// TwinCAT 3 PLC project PRG_PLCHMIManager
// Title: B_PLCHMIManager
// Company: RafalOS
// Author: Rafał Osajda
// ProjectVersion: 0.0.0.23
// ProgramVersion: 3.1.4024.0
// CompilerDefines: VISU_USEWSTRING
// libraries:
//   B_Base, * (RafalOS)
//   B_Base_HMI_Connector, * (RafalOS)
//   B_HMIElements, * (RafalOS)
//   B_HMIManager, * (RafałOS)
//   B_MachineControl_HMI_Connector, * (RafalOS)
//   B_StatesAndModes, * (RafalOS)
//   CmpBitmapPool, * (System)
//   Tc2_Standard, * (Beckhoff Automation GmbH)
//   Tc2_System, * (Beckhoff Automation GmbH)
//   Tc3_Module, * (Beckhoff Automation GmbH)
//   VisuDialogs, * (System)
//   VisuSymbols,3.5.10.0,System
// project tree:
//   / GlobalTextList.TcGTLO, PlcTask.TcTTO, Visualization Manager.TcVMO (not stored), VISU_TASK.TcTTO
//   POUs/ MAIN.TcPOU
//   VISUs/Dialogs/ D_AddRecipe.TcVIS, D_DeleteRecipeCleim.TcVIS
//   VISUs/Frame/ F_Descriptor.TcVIS, F_DiagramState.TcVIS
//   VISUs/Graphics/ ImagePool.TcIPO (not stored)
//   VISUs/Keyboards/ KlawiaturaCyfry.TcVIS, KlawiaturaLitery.TcVIS
//   VISUs/ MainFrame.TcVIS, TextListGlobal.TcTLO, Visualization.TcVIS
//   VISUs/MainMenuFrame/ F_00_MainScreen.TcVIS, F_01_Parameters.TcVIS, F_02_Recipe.TcVIS, F_03_Events.TcVIS, F_04_ChangeMode.TcVIS, F_05_Statistics.TcVIS, F_06_Diagram.TcVIS, F_07_Settings.TcVIS
//   VISUs/MainMenu/ F_MainMenu_00.TcVIS, F_MainMenu_01.TcVIS, F_MainMenu_02.TcVIS, F_MainMenu_03.TcVIS, F_MainMenu_04.TcVIS, F_MainMenu_05.TcVIS, F_MainMenu_06.TcVIS, F_MainMenu_07.TcVIS
//   VISUs/TextListFrame/ TextList_00.TcTLO, TextList_01.TcTLO, TextList_02.TcTLO, TextList_03.TcTLO, TextList_04.TcTLO, TextList_05.TcTLO, TextList_06.TcTLO, TextList_07.TcTLO
// real-time tasks:
//   TASK PlcTask: cycle T#10ms, priority 20, ADS port 350
//   TASK VISU_TASK: cycle T#200000us, priority 30, ADS port 351

CONFIGURATION PRG_PLCHMIManager
    RESOURCE PLC ON TwinCAT3
        TASK PlcTask(INTERVAL := T#10ms, PRIORITY := 20);
        TASK VISU_TASK(INTERVAL := T#200000us, PRIORITY := 30);
        PROGRAM MAIN WITH PlcTask : MAIN;
        PROGRAM VisuElems_Visu_Prg WITH VISU_TASK : VisuElems.Visu_Prg;
    END_RESOURCE
END_CONFIGURATION

// ---- POUs/MAIN.TcPOU
PROGRAM MAIN
VAR
	stDataHMI : ST_HMIManager;
END_VAR

END_PROGRAM

// ---- GlobalTextList.TcGTLO
TEXTLIST GlobalTextList
  338 = '!'
  340 = '"'
  991 = '#'
  344 = '$'
  346 = '%'
  858 = '%d'
  949 = '%s'
  399 = '%s sfdasgfds gkds gow gk wjd k gj dlkg jdl glkd sj g ld jdlgj lg lsdg'
  169 = '&'
  992 = "'"
  174 = '('
  634 = ')'
  333 = '*'
  332 = '+'
  90 = '+/-'
  153 = ','
  157 = '-'
  43 = '-Wartoscdomyślna: %s'
  155 = '.'
  171 = '/'
  179 = '0'
  337 = '1'
  339 = '2'
  341 = '3'
  343 = '4'
  345 = '5'
  347 = '6'
  170 = '7'
  172 = '8'
  176 = '9'
  156 = ':'
  154 = ';'
  137 = '<'
  181 = '='
  138 = '>'
  184 = '?'
  993 = '@'
  160 = 'a'
  161 = 'A'
  834 = 'Abort'
  147 = 'b'
  148 = 'B'
  781 = 'Back'
  92 = 'Backspace'
  143 = 'c'
  144 = 'C'
  987 = 'CANCEL'
  131 = 'Change Mode'
  780 = 'Clear'
  164 = 'd'
  974 = 'D'
  300 = 'DE'
  243 = 'Diagram'
  30 = 'Domyślna : %s'
  801 = 'Domyślna wartość : %s'
  998 = 'e'
  999 = 'E'
  477 = 'EN'
  779 = 'ESC'
  975 = 'f'
  976 = 'F'
  977 = 'g'
  978 = 'G'
  979 = 'h'
  980 = 'H'
  970 = 'Hold'
  1008 = 'i'
  1009 = 'I'
  981 = 'j'
  982 = 'J'
  791 = 'Jedn.'
  388 = 'Jednostka'
  983 = 'k'
  984 = 'K'
  985 = 'l'
  986 = 'L'
  151 = 'm'
  152 = 'M'
  1175 = 'Max :'
  192 = 'Max:'
  55 = 'Max: %s'
  690 = 'Min :'
  191 = 'Min:'
  1119 = 'Min: %s'
  149 = 'n'
  150 = 'N'
  1010 = 'o'
  1011 = 'O'
  778 = 'OK'
  623 = 'Okno główne'
  1328 = 'Opis'
  1012 = 'p'
  1013 = 'P'
  689 = 'Parametry'
  281 = 'PL'
  461 = 'q'
  995 = 'Q'
  1000 = 'r'
  1001 = 'R'
  994 = 'Receptury'
  444 = 'Reset'
  162 = 's'
  163 = 'S'
  936 = 'Settings'
  782 = 'Shift'
  783 = 'Space'
  613 = 'Start'
  81 = 'Statistics'
  745 = 'Stop'
  96 = 'Suspend'
  1002 = 't'
  1003 = 'T'
  1006 = 'u'
  1007 = 'U'
  708 = 'UnHold'
  950 = 'UnSuspend'
  145 = 'v'
  146 = 'V'
  996 = 'w'
  997 = 'W'
  1118 = 'Wartość'
  141 = 'x'
  142 = 'X'
  139 = 'y'
  140 = 'Y'
  1004 = 'z'
  1005 = 'Z'
  829 = 'Zdarzenia'
  787 = '['
  187 = '\\'
  788 = ']'
  335 = '^'
  158 = '_'
  239 = '_aktualny stan'
  803 = '_aktualny tryb'
  175 = '_anuluj'
  370 = '_brak receptury'
  391 = '_całkowity czas'
  1244 = '_czas pracy w trybie'
  1278 = '_dostępne tryby'
  1014 = '_ostrzeżenie'
  159 = '_pokaz czasy'
  312 = '_przywrócdomyślną'
  988 = '_utworz'
  1089 = '_utworzszbalony'
  1214 = '_wartoscdomyślna '
  1108 = '_wartoscdomyślna: %s'
  667 = '_wartość'
  411 = '_wybierz jezyk'
  1043 = '_zapisz'
  1087 = '_zmien tryb'
  786 = '{'
  790 = '|'
  789 = '}'
  334 = '~'
  186 = '´'
END_TEXTLIST

// ---- VISUs/Dialogs/D_AddRecipe.TcVIS
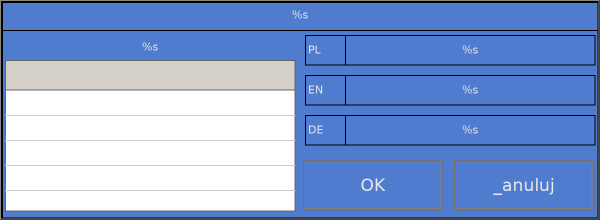
VISUALIZATION D_AddRecipe  // 600x220
VAR_IN_OUT
	{attribute "VAR_IN_OUT_AS_POINTER}
	stData		: ST_MCHMIPrepareScreen_02_XX_AddRecipe;
END_VAR
    Rectangle (0,0 600x220)
    Rectangle (305,35 290x30), "PL"
    Line (0,30) (600,30)
    Rectangle (3,3 594x24), "%s", text variable: stData.wsTitle
    Button (454,160 140x50), "_anuluj", text list: 'TextListGlobal', text index: 2
        OnMouseDown: execute { stData.bCancel := TRUE; }
        OnMouseUp: CloseDialog Dialog=D_AddRecipe, Result=Ignore, NumpadKeypadSet=True
    Button (303,160 140x50), "OK"
        OnMouseDown: execute { stData.bOk := TRUE; }
        OnMouseUp: CloseDialog Dialog=D_AddRecipe, Result=OK, NumpadKeypadSet=True
    Rectangle (345,35 250x30), "%s", text variable: stData.stNewNames.arrText [1]
        OnMouseDown: write the text variable via KlawiaturaLitery
    Rectangle (305,75 290x30), "EN"
    Rectangle (345,75 250x30), "%s", text variable: stData.stNewNames.arrText [2]
        OnMouseDown: write the text variable via KlawiaturaLitery
    Rectangle (305,115 290x30), "DE"
    Rectangle (345,115 250x30), "%s", text variable: stData.stNewNames.arrText [3]
        OnMouseDown: write the text variable via KlawiaturaLitery
    Rectangle (3,35 294x24), "%s", text variable: stData.wsSource
    Table (5,60 290x151), data array: stData.arrListOfName
        p3854506369: stData.arrListOfName[INDEX]
        p1128707560: stData.iNumberOfNames
        p1822360349: stData.bSelectedRow
        p1137915858: stData.iSelectedName
END_VISUALIZATION

// ---- VISUs/Dialogs/D_DeleteRecipeCleim.TcVIS
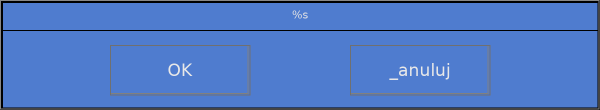
VISUALIZATION D_DeleteRecipeCleim  // 600x110
VAR_IN_OUT
	stData : ST_MCHMIPrepareScreen_02_XX_DeleteRecipe;
END_VAR
    Rectangle (0,0 600x110)
    Line (0,30) (600,30)
    Rectangle (3,3 594x24), "%s", text variable: stData.wsNameRecipe, text list: 'TextList_02', text index: 0
    Button (350,45 140x50), "_anuluj", text list: 'TextListGlobal', text index: 2
        OnMouseDown: execute { stData.bCancel := TRUE; }
        OnMouseUp: CloseDialog Dialog=D_DeleteRecipeCleim, Result=Ignore, NumpadKeypadSet=True
    Button (110,45 140x50), "OK"
        OnMouseDown: execute { stData.bOK := TRUE; }
        OnMouseUp: CloseDialog Dialog=D_DeleteRecipeCleim, Result=OK, NumpadKeypadSet=True
END_VISUALIZATION

// ---- VISUs/Frame/F_Descriptor.TcVIS
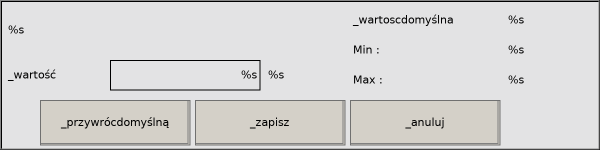
VISUALIZATION F_Descriptor  // 600x150
VAR_IN_OUT
	stData 	: ST_BaseHMIDescriptorEdit;
END_VAR
    Rectangle (0,0 600x150)
    Rectangle (5,5 330x50), "%s", text variable: stData.wsText
    Rectangle (350,35 100x30), "Min :"
    Rectangle (350,65 100x30), "Max :"
    Rectangle (350,5 150x30), "_wartoscdomyślna", text list: 'TextListGlobal', text index: 5
    Rectangle (505,5 50x30), "%s", text variable: stData.rDefaultValue, text list: 'TextList_02', text index: 1
    Rectangle (505,35 50x30), "%s", text variable: stData.rMin
    Rectangle (505,65 50x30), "%s", text variable: stData.rMax
    Rectangle (5,60 100x30), "_wartość", text list: 'TextListGlobal', text index: 6
    Rectangle (110,60 150x30), "%s", text variable: stData.rValue
        OnMouseDown: write the text variable via KlawiaturaCyfry, min stData.rMin, max stData.rMax
    Rectangle (265,60 70x30), "%s", text variable: stData.sUnit
    Button (40,100 150x45), "_przywrócdomyślną", invisible if: not stData.bVisibleSetDefault, text list: 'TextListGlobal', text index: 3
        OnMouseDown: execute { stData.bSetDefault := TRUE; }
    Button (195,100 150x45), "_zapisz", invisible if: not stData.bVisibleSave, text list: 'TextListGlobal', text index: 4
        OnMouseDown: execute { stData.bSave := TRUE; }
    Button (350,100 150x45), "_anuluj", invisible if: not stData.bVisibleCancel, text list: 'TextListGlobal', text index: 2
        OnMouseDown: execute { stData.bCancel := TRUE; }
END_VISUALIZATION

// ---- VISUs/Frame/F_DiagramState.TcVIS
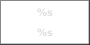
VISUALIZATION F_DiagramState  // 90x45
VAR_IN_OUT
	stStateInfo		: ST_MCHMIPrepareScreen_06_XX_State;
END_VAR
    Rectangle (0,0 90x45), colour variable: stStateInfo.dwBackgroud
        p1271844420: stStateInfo.iWidthFrame
    Rectangle (5,5 80x15), "%s", text variable: stStateInfo.wsNameOfState
    Rectangle (5,25 80x15), "%s", text variable: stStateInfo.sTime, invisible if: not stStateInfo.bShowTime
END_VISUALIZATION

// ---- VISUs/Keyboards/KlawiaturaCyfry.TcVIS
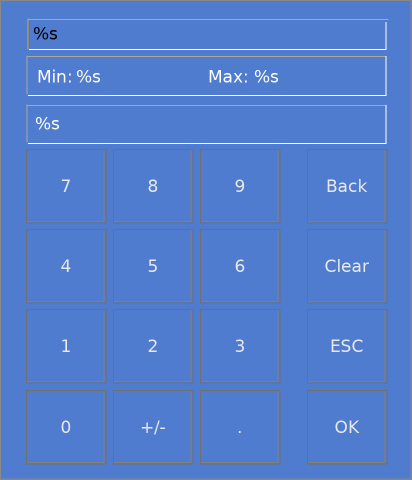
VISUALIZATION KlawiaturaCyfry  // 412x480
VAR_INPUT
	stVariableValue : STRING;
	stMin : STRING;
	stMax : STRING;
	stTitle : STRING;
	flags : DWORD;
END_VAR
VAR
	bInit : BOOL;
	stMessage : STRING;
	stOutputValue : STRING;
END_VAR
    Rectangle (0,0 412x480)
    Rectangle (10,142 393x83)
    Rectangle (10,225 393x80)
    Rectangle (10,305 393x80)
    Rectangle (10,385 393x85)
    Button (307,390 80x74), "OK"
        OnMouseDown: CloseDialog Dialog=KlawiaturaCyfry, Result=OK, NumpadKeypad=True, NumpadKeypadSet=True
    Button (307,309 80x74), "ESC"
        OnMouseDown: CloseDialog Dialog=KlawiaturaCyfry, Result=Cancel, NumpadKeypad=True, NumpadKeypadSet=True
    Button (307,229 80x74), "Clear"
        OnMouseDown: execute {
            stVariableValue := '';
            stOutputValue := '';
            flags := flags AND 16#0008;
            flags := flags AND 16#0010;
        }
    Button (307,149 80x74), "Back"
        OnMouseDown: execute { VisuDlg_CheckedBack(stOutputValue, stVariableValue, bInit); }
    Button (200,390 80x74), "."
        OnMouseDown: execute { VisuDlg_CheckedAppend(stOutputValue, stVariableValue, bInit, (flags AND VisuElems.Visu_InputFlags.Password) = 1, '.'); }
    Button (113,390 80x74), "+/-"
        OnMouseDown: execute { VisuDlg_CheckedChangeSign(stOutputValue, stVariableValue, bInit, (flags AND VisuElems.Visu_InputFlags.Password) = 1); }
    Button (26,390 80x74), "0"
        OnMouseDown: execute { VisuDlg_CheckedAppend(stOutputValue, stVariableValue, bInit, (flags AND VisuElems.Visu_InputFlags.Password) = 1, '0'); }
    Button (26,309 80x74), "1"
        OnMouseDown: execute { VisuDlg_CheckedAppend(stOutputValue, stVariableValue, bInit, (flags AND VisuElems.Visu_InputFlags.Password) = 1, '1'); }
    Button (113,309 80x74), "2"
        OnMouseDown: execute { VisuDlg_CheckedAppend(stOutputValue, stVariableValue, bInit, (flags AND VisuElems.Visu_InputFlags.Password) = 1, '2'); }
    Button (200,309 80x74), "3"
        OnMouseDown: execute { VisuDlg_CheckedAppend(stOutputValue, stVariableValue, bInit, (flags AND VisuElems.Visu_InputFlags.Password) = 1, '3'); }
    Button (26,229 80x74), "4"
        OnMouseDown: execute { VisuDlg_CheckedAppend(stOutputValue, stVariableValue, bInit, (flags AND VisuElems.Visu_InputFlags.Password) = 1, '4'); }
    Button (113,229 80x74), "5"
        OnMouseDown: execute { VisuDlg_CheckedAppend(stOutputValue, stVariableValue, bInit, (flags AND VisuElems.Visu_InputFlags.Password) = 1, '5'); }
    Button (200,229 80x74), "6"
        OnMouseDown: execute { VisuDlg_CheckedAppend(stOutputValue, stVariableValue, bInit, (flags AND VisuElems.Visu_InputFlags.Password) = 1, '6'); }
    Button (26,149 80x74), "7"
        OnMouseDown: execute { VisuDlg_CheckedAppend(stOutputValue, stVariableValue, bInit, (flags AND VisuElems.Visu_InputFlags.Password) = 1, '7'); }
    Button (113,149 80x74), "8"
        OnMouseDown: execute { VisuDlg_CheckedAppend(stOutputValue, stVariableValue, bInit, (flags AND VisuElems.Visu_InputFlags.Password) = 1, '8'); }
    Button (200,149 80x74), "9"
        OnMouseDown: execute { VisuDlg_CheckedAppend(stOutputValue, stVariableValue, bInit, (flags AND VisuElems.Visu_InputFlags.Password) = 1, '9'); }
    Rectangle (10,10 393x48)
    Rectangle (10,57 393x85)
    Rectangle (73,64 127x25), "%s", text variable: stMin, invisible if: LEN(stMin) = 0
    Rectangle (251,64 127x25), "%s", text variable: stMax, invisible if: LEN(stMax) = 0
    Rectangle (205,64 45x25), "Max:", text variable: stMin, invisible if: LEN(stMax) = 0
        p55702900: SEL(((UDINT_TO_DINT(flags AND 16#0010))=16#0010),16#FF000000,16#FFFF0000)
    Rectangle (402,470 4x4)
    Polyline (27,94) (27,56) (385,56)
    Polyline (27,142) (27,105) (385,105)
    Polyline (28,49) (28,19) (388,19)
    Polyline (28,143) (386,143) (386,105)
    Polyline (28,95) (386,95) (386,56)
    Polyline (29,49) (386,49) (386,21)
    Polyline (29,48) (29,21) (386,21)
    Rectangle (32,111 349x25), "%s", text variable: stMessage
    Rectangle (34,64 41x25), "Min:", text variable: stMin, invisible if: LEN(stMin) = 0
        p55702900: SEL(((UDINT_TO_DINT(flags AND 16#0008))=16#0008),16#FF000000,16#FFFF0000)
    Rectangle (30,21 355x25), "%s", text variable: stOutputValue
END_VISUALIZATION

// ---- VISUs/Keyboards/KlawiaturaLitery.TcVIS
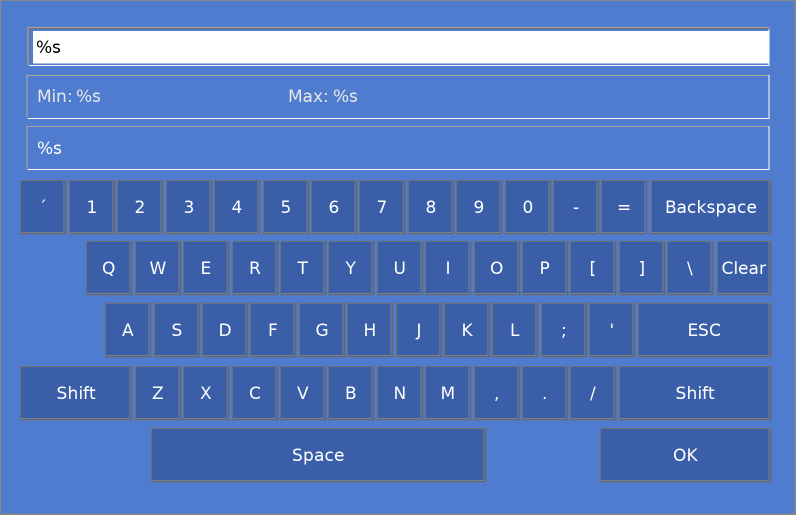
VISUALIZATION KlawiaturaLitery  // 796x515
VAR_INPUT
	stVariableValue : STRING;
	stMin : STRING;
	stMax : STRING;
	stTitle : STRING;
	flags : DWORD;
END_VAR
VAR
	bInit : BOOL;
	bShift : BOOL;
	stMessage : STRING;
	stOutputValue : STRING;
END_VAR
    Rectangle (0,0 796x515)
    Rectangle (12,169 773x70)
    Rectangle (12,240 773x62)
    Rectangle (12,301 773x63)
    Rectangle (12,364 773x62)
    Rectangle (12,423 773x75)
    Button (600,428 171x54), "OK"
        OnMouseDown: CloseDialog Dialog=KlawiaturaLitery, Result=OK, NumpadKeypad=True, NumpadKeypadSet=True
    Button (638,303 133x54), "ESC"
        OnMouseDown: CloseDialog Dialog=KlawiaturaLitery, Result=Cancel, NumpadKeypad=True, NumpadKeypadSet=True
    Button (717,241 54x54), "Clear"
        OnMouseDown: execute { stVariableValue := ''; stOutputValue := ''; }
    Button (651,180 120x54), "Backspace"
        OnMouseDown: execute { VisuDlg_CheckedBack(stOutputValue, stVariableValue, bInit); }
    Button (619,366 152x54), "Shift"
        OnMouseDown: toggle bShift
    Button (151,428 335x54), "Space"
        OnMouseDown: execute { VisuDlg_CheckedAppend(stOutputValue, stVariableValue, bInit, (flags AND VisuElems.Visu_InputFlags.Password) = 1, ' '); }
    Button (667,241 46x54), "|", invisible if: NOT bShift
        OnMouseDown: execute { VisuDlg_CheckedAppend(stOutputValue, stVariableValue, bInit, (flags AND VisuElems.Visu_InputFlags.Password) = 1, '|'); }
    Button (474,366 46x54), "<", invisible if: NOT bShift
        OnMouseDown: execute { VisuDlg_CheckedAppend(stOutputValue, stVariableValue, bInit, (flags AND VisuElems.Visu_InputFlags.Password) = 1, '<'); }
    Button (522,366 46x54), ">", invisible if: NOT bShift
        OnMouseDown: execute { VisuDlg_CheckedAppend(stOutputValue, stVariableValue, bInit, (flags AND VisuElems.Visu_InputFlags.Password) = 1, '>'); }
    Button (328,241 46x54), "y", invisible if: NOT bShift
        OnMouseDown: execute { VisuDlg_CheckedAppend(stOutputValue, stVariableValue, bInit, (flags AND VisuElems.Visu_InputFlags.Password) = 1, 'y'); }
    Button (328,241 46x54), "Y", invisible if: bShift
        OnMouseDown: execute { VisuDlg_CheckedAppend(stOutputValue, stVariableValue, bInit, (flags AND VisuElems.Visu_InputFlags.Password) = 1, 'Y'); }
    Button (183,366 46x54), "x", invisible if: NOT bShift
        OnMouseDown: execute { VisuDlg_CheckedAppend(stOutputValue, stVariableValue, bInit, (flags AND VisuElems.Visu_InputFlags.Password) = 1, 'x'); }
    Button (183,366 46x54), "X", invisible if: bShift
        OnMouseDown: execute { VisuDlg_CheckedAppend(stOutputValue, stVariableValue, bInit, (flags AND VisuElems.Visu_InputFlags.Password) = 1, 'X'); }
    Button (232,366 46x54), "c", invisible if: NOT bShift
        OnMouseDown: execute { VisuDlg_CheckedAppend(stOutputValue, stVariableValue, bInit, (flags AND VisuElems.Visu_InputFlags.Password) = 1, 'c'); }
    Button (232,366 46x54), "C", invisible if: bShift
        OnMouseDown: execute { VisuDlg_CheckedAppend(stOutputValue, stVariableValue, bInit, (flags AND VisuElems.Visu_InputFlags.Password) = 1, 'C'); }
    Button (280,366 46x54), "v", invisible if: NOT bShift
        OnMouseDown: execute { VisuDlg_CheckedAppend(stOutputValue, stVariableValue, bInit, (flags AND VisuElems.Visu_InputFlags.Password) = 1, 'v'); }
    Button (280,366 46x54), "V", invisible if: bShift
        OnMouseDown: execute { VisuDlg_CheckedAppend(stOutputValue, stVariableValue, bInit, (flags AND VisuElems.Visu_InputFlags.Password) = 1, 'V'); }
    Button (328,366 46x54), "b", invisible if: NOT bShift
        OnMouseDown: execute { VisuDlg_CheckedAppend(stOutputValue, stVariableValue, bInit, (flags AND VisuElems.Visu_InputFlags.Password) = 1, 'b'); }
    Button (328,366 46x54), "B", invisible if: bShift
        OnMouseDown: execute { VisuDlg_CheckedAppend(stOutputValue, stVariableValue, bInit, (flags AND VisuElems.Visu_InputFlags.Password) = 1, 'B'); }
    Button (377,366 46x54), "n", invisible if: NOT bShift
        OnMouseDown: execute { VisuDlg_CheckedAppend(stOutputValue, stVariableValue, bInit, (flags AND VisuElems.Visu_InputFlags.Password) = 1, 'n'); }
    Button (377,366 46x54), "N", invisible if: bShift
        OnMouseDown: execute { VisuDlg_CheckedAppend(stOutputValue, stVariableValue, bInit, (flags AND VisuElems.Visu_InputFlags.Password) = 1, 'N'); }
    Button (425,366 46x54), "m", invisible if: NOT bShift
        OnMouseDown: execute { VisuDlg_CheckedAppend(stOutputValue, stVariableValue, bInit, (flags AND VisuElems.Visu_InputFlags.Password) = 1, 'm'); }
    Button (425,366 46x54), "M", invisible if: bShift
        OnMouseDown: execute { VisuDlg_CheckedAppend(stOutputValue, stVariableValue, bInit, (flags AND VisuElems.Visu_InputFlags.Password) = 1, 'M'); }
    Button (541,303 46x54), ":", invisible if: NOT bShift
        OnMouseDown: execute { VisuDlg_CheckedAppend(stOutputValue, stVariableValue, bInit, (flags AND VisuElems.Visu_InputFlags.Password) = 1, ':'); }
    Button (553,180 46x54), "_", invisible if: NOT bShift
        OnMouseDown: execute { VisuDlg_CheckedAppend(stOutputValue, stVariableValue, bInit, (flags AND VisuElems.Visu_InputFlags.Password) = 1, '_'); }
    Button (105,303 46x54), "a", invisible if: NOT bShift
        OnMouseDown: execute { VisuDlg_CheckedAppend(stOutputValue, stVariableValue, bInit, (flags AND VisuElems.Visu_InputFlags.Password) = 1, 'a'); }
    Button (105,303 46x54), "A", invisible if: bShift
        OnMouseDown: execute { VisuDlg_CheckedAppend(stOutputValue, stVariableValue, bInit, (flags AND VisuElems.Visu_InputFlags.Password) = 1, 'A'); }
    Button (154,303 46x54), "s", invisible if: NOT bShift
        OnMouseDown: execute { VisuDlg_CheckedAppend(stOutputValue, stVariableValue, bInit, (flags AND VisuElems.Visu_InputFlags.Password) = 1, 's'); }
    Button (154,303 46x54), "S", invisible if: bShift
        OnMouseDown: execute { VisuDlg_CheckedAppend(stOutputValue, stVariableValue, bInit, (flags AND VisuElems.Visu_InputFlags.Password) = 1, 'S'); }
    Button (202,303 46x54), "d", invisible if: NOT bShift
        OnMouseDown: execute { VisuDlg_CheckedAppend(stOutputValue, stVariableValue, bInit, (flags AND VisuElems.Visu_InputFlags.Password) = 1, 'd'); }
    Button (202,303 46x54), "D", invisible if: bShift
        OnMouseDown: execute { VisuDlg_CheckedAppend(stOutputValue, stVariableValue, bInit, (flags AND VisuElems.Visu_InputFlags.Password) = 1, 'D'); }
    Button (250,303 46x54), "f", invisible if: NOT bShift
        OnMouseDown: execute { VisuDlg_CheckedAppend(stOutputValue, stVariableValue, bInit, (flags AND VisuElems.Visu_InputFlags.Password) = 1, 'f'); }
    Button (250,303 46x54), "F", invisible if: bShift
        OnMouseDown: execute { VisuDlg_CheckedAppend(stOutputValue, stVariableValue, bInit, (flags AND VisuElems.Visu_InputFlags.Password) = 1, 'F'); }
    Button (299,303 46x54), "g", invisible if: NOT bShift
        OnMouseDown: execute { VisuDlg_CheckedAppend(stOutputValue, stVariableValue, bInit, (flags AND VisuElems.Visu_InputFlags.Password) = 1, 'g'); }
    Button (299,303 46x54), "G", invisible if: bShift
        OnMouseDown: execute { VisuDlg_CheckedAppend(stOutputValue, stVariableValue, bInit, (flags AND VisuElems.Visu_InputFlags.Password) = 1, 'G'); }
    Button (347,303 46x54), "h", invisible if: NOT bShift
        OnMouseDown: execute { VisuDlg_CheckedAppend(stOutputValue, stVariableValue, bInit, (flags AND VisuElems.Visu_InputFlags.Password) = 1, 'h'); }
    Button (347,303 46x54), "H", invisible if: bShift
        OnMouseDown: execute { VisuDlg_CheckedAppend(stOutputValue, stVariableValue, bInit, (flags AND VisuElems.Visu_InputFlags.Password) = 1, 'H'); }
    Button (396,303 46x54), "j", invisible if: NOT bShift
        OnMouseDown: execute { VisuDlg_CheckedAppend(stOutputValue, stVariableValue, bInit, (flags AND VisuElems.Visu_InputFlags.Password) = 1, 'j'); }
    Button (396,303 46x54), "J", invisible if: bShift
        OnMouseDown: execute { VisuDlg_CheckedAppend(stOutputValue, stVariableValue, bInit, (flags AND VisuElems.Visu_InputFlags.Password) = 1, 'J'); }
    Button (444,303 46x54), "k", invisible if: NOT bShift
        OnMouseDown: execute { VisuDlg_CheckedAppend(stOutputValue, stVariableValue, bInit, (flags AND VisuElems.Visu_InputFlags.Password) = 1, 'k'); }
    Button (444,303 46x54), "K", invisible if: bShift
        OnMouseDown: execute { VisuDlg_CheckedAppend(stOutputValue, stVariableValue, bInit, (flags AND VisuElems.Visu_InputFlags.Password) = 1, 'K'); }
    Button (492,303 46x54), "l", invisible if: NOT bShift
        OnMouseDown: execute { VisuDlg_CheckedAppend(stOutputValue, stVariableValue, bInit, (flags AND VisuElems.Visu_InputFlags.Password) = 1, 'l'); }
    Button (492,303 46x54), "L", invisible if: bShift
        OnMouseDown: execute { VisuDlg_CheckedAppend(stOutputValue, stVariableValue, bInit, (flags AND VisuElems.Visu_InputFlags.Password) = 1, 'L'); }
    Button (166,180 46x54), "#", invisible if: NOT bShift
        OnMouseDown: execute { VisuDlg_CheckedAppend(stOutputValue, stVariableValue, bInit, (flags AND VisuElems.Visu_InputFlags.Password) = 1, '#'); }
    Button (117,180 46x54), "@", invisible if: NOT bShift
        OnMouseDown: execute { VisuDlg_CheckedAppend(stOutputValue, stVariableValue, bInit, (flags AND VisuElems.Visu_InputFlags.Password) = 1, '@'); }
    Button (86,241 46x54), "q", invisible if: NOT bShift
        OnMouseDown: execute { VisuDlg_CheckedAppend(stOutputValue, stVariableValue, bInit, (flags AND VisuElems.Visu_InputFlags.Password) = 1, 'q'); }
    Button (86,241 46x54), "Q", invisible if: bShift
        OnMouseDown: execute { VisuDlg_CheckedAppend(stOutputValue, stVariableValue, bInit, (flags AND VisuElems.Visu_InputFlags.Password) = 1, 'Q'); }
    Button (135,241 46x54), "w", invisible if: NOT bShift
        OnMouseDown: execute { VisuDlg_CheckedAppend(stOutputValue, stVariableValue, bInit, (flags AND VisuElems.Visu_InputFlags.Password) = 1, 'w'); }
    Button (135,241 46x54), "W", invisible if: bShift
        OnMouseDown: execute { VisuDlg_CheckedAppend(stOutputValue, stVariableValue, bInit, (flags AND VisuElems.Visu_InputFlags.Password) = 1, 'W'); }
    Button (183,241 46x54), "e", invisible if: NOT bShift
        OnMouseDown: execute { VisuDlg_CheckedAppend(stOutputValue, stVariableValue, bInit, (flags AND VisuElems.Visu_InputFlags.Password) = 1, 'e'); }
    Button (183,241 46x54), "E", invisible if: bShift
        OnMouseDown: execute { VisuDlg_CheckedAppend(stOutputValue, stVariableValue, bInit, (flags AND VisuElems.Visu_InputFlags.Password) = 1, 'E'); }
    Button (232,241 46x54), "r", invisible if: NOT bShift
        OnMouseDown: execute { VisuDlg_CheckedAppend(stOutputValue, stVariableValue, bInit, (flags AND VisuElems.Visu_InputFlags.Password) = 1, 'r'); }
    Button (232,241 46x54), "R", invisible if: bShift
        OnMouseDown: execute { VisuDlg_CheckedAppend(stOutputValue, stVariableValue, bInit, (flags AND VisuElems.Visu_InputFlags.Password) = 1, 'R'); }
    Button (280,241 46x54), "t", invisible if: NOT bShift
        OnMouseDown: execute { VisuDlg_CheckedAppend(stOutputValue, stVariableValue, bInit, (flags AND VisuElems.Visu_InputFlags.Password) = 1, 't'); }
    Button (280,241 46x54), "T", invisible if: bShift
        OnMouseDown: execute { VisuDlg_CheckedAppend(stOutputValue, stVariableValue, bInit, (flags AND VisuElems.Visu_InputFlags.Password) = 1, 'T'); }
    Button (135,366 46x54), "z", invisible if: NOT bShift
        OnMouseDown: execute { VisuDlg_CheckedAppend(stOutputValue, stVariableValue, bInit, (flags AND VisuElems.Visu_InputFlags.Password) = 1, 'z'); }
    Button (135,366 46x54), "Z", invisible if: bShift
        OnMouseDown: execute { VisuDlg_CheckedAppend(stOutputValue, stVariableValue, bInit, (flags AND VisuElems.Visu_InputFlags.Password) = 1, 'Z'); }
    Button (377,241 46x54), "u", invisible if: NOT bShift
        OnMouseDown: execute { VisuDlg_CheckedAppend(stOutputValue, stVariableValue, bInit, (flags AND VisuElems.Visu_InputFlags.Password) = 1, 'u'); }
    Button (377,241 46x54), "U", invisible if: bShift
        OnMouseDown: execute { VisuDlg_CheckedAppend(stOutputValue, stVariableValue, bInit, (flags AND VisuElems.Visu_InputFlags.Password) = 1, 'U'); }
    Button (425,241 46x54), "i", invisible if: NOT bShift
        OnMouseDown: execute { VisuDlg_CheckedAppend(stOutputValue, stVariableValue, bInit, (flags AND VisuElems.Visu_InputFlags.Password) = 1, 'i'); }
    Button (425,241 46x54), "I", invisible if: bShift
        OnMouseDown: execute { VisuDlg_CheckedAppend(stOutputValue, stVariableValue, bInit, (flags AND VisuElems.Visu_InputFlags.Password) = 1, 'I'); }
    Button (474,241 46x54), "o", invisible if: NOT bShift
        OnMouseDown: execute { VisuDlg_CheckedAppend(stOutputValue, stVariableValue, bInit, (flags AND VisuElems.Visu_InputFlags.Password) = 1, 'o'); }
    Button (474,241 46x54), "O", invisible if: bShift
        OnMouseDown: execute { VisuDlg_CheckedAppend(stOutputValue, stVariableValue, bInit, (flags AND VisuElems.Visu_InputFlags.Password) = 1, 'O'); }
    Button (522,241 46x54), "p", invisible if: NOT bShift
        OnMouseDown: execute { VisuDlg_CheckedAppend(stOutputValue, stVariableValue, bInit, (flags AND VisuElems.Visu_InputFlags.Password) = 1, 'p'); }
    Button (522,241 46x54), "P", invisible if: bShift
        OnMouseDown: execute { VisuDlg_CheckedAppend(stOutputValue, stVariableValue, bInit, (flags AND VisuElems.Visu_InputFlags.Password) = 1, 'P'); }
    Button (601,180 46x54), "+", invisible if: NOT bShift
        OnMouseDown: execute { VisuDlg_CheckedAppend(stOutputValue, stVariableValue, bInit, (flags AND VisuElems.Visu_InputFlags.Password) = 1, '+'); }
    Button (408,180 46x54), "*", invisible if: NOT bShift
        OnMouseDown: execute { VisuDlg_CheckedAppend(stOutputValue, stVariableValue, bInit, (flags AND VisuElems.Visu_InputFlags.Password) = 1, '*'); }
    Button (20,180 46x54), "~", invisible if: NOT bShift
        OnMouseDown: execute { VisuDlg_CheckedAppend(stOutputValue, stVariableValue, bInit, (flags AND VisuElems.Visu_InputFlags.Password) = 1, '~'); }
    Button (311,180 46x54), "^", invisible if: NOT bShift
        OnMouseDown: execute { VisuDlg_CheckedAppend(stOutputValue, stVariableValue, bInit, (flags AND VisuElems.Visu_InputFlags.Password) = 1, '^'); }
    Button (69,180 46x54), "!", invisible if: NOT bShift
        OnMouseDown: execute { VisuDlg_CheckedAppend(stOutputValue, stVariableValue, bInit, (flags AND VisuElems.Visu_InputFlags.Password) = 1, '!'); }
    Button (589,303 46x54), """, invisible if: NOT bShift
        OnMouseDown: execute { VisuDlg_CheckedAppend(stOutputValue, stVariableValue, bInit, (flags AND VisuElems.Visu_InputFlags.Password) = 1, '"'); }
    Button (214,180 46x54), "$", invisible if: NOT bShift
        OnMouseDown: execute { VisuDlg_CheckedAppend(stOutputValue, stVariableValue, bInit, (flags AND VisuElems.Visu_InputFlags.Password) = 1, '$$'); }
    Button (263,180 46x54), "%", invisible if: NOT bShift
        OnMouseDown: execute { VisuDlg_CheckedAppend(stOutputValue, stVariableValue, bInit, (flags AND VisuElems.Visu_InputFlags.Password) = 1, '%'); }
    Button (359,180 46x54), "&", invisible if: NOT bShift
        OnMouseDown: execute { VisuDlg_CheckedAppend(stOutputValue, stVariableValue, bInit, (flags AND VisuElems.Visu_InputFlags.Password) = 1, '&'); }
    Button (456,180 46x54), "(", invisible if: NOT bShift
        OnMouseDown: execute { VisuDlg_CheckedAppend(stOutputValue, stVariableValue, bInit, (flags AND VisuElems.Visu_InputFlags.Password) = 1, '('); }
    Button (505,180 46x54), ")", invisible if: NOT bShift
        OnMouseDown: execute { VisuDlg_CheckedAppend(stOutputValue, stVariableValue, bInit, (flags AND VisuElems.Visu_InputFlags.Password) = 1, ')'); }
    Button (570,366 46x54), "?", invisible if: NOT bShift
        OnMouseDown: execute { VisuDlg_CheckedAppend(stOutputValue, stVariableValue, bInit, (flags AND VisuElems.Visu_InputFlags.Password) = 1, '?'); }
    Rectangle (12,72 773x97)
    Rectangle (34,132 734x32), "%s", text variable: stMessage
    Rectangle (12,10 773x62)
    Polyline (27,169) (27,126) (769,126)
    Polyline (27,118) (27,75) (769,75)
    Polyline (28,65) (28,27) (769,27)
    Polyline (28,169) (769,169) (769,126)
    Polyline (28,118) (769,118) (769,75)
    Polyline (29,65) (769,65) (769,28)
    Polyline (29,63) (29,28) (769,28)
    Rectangle (33,31 736x32), "%s", text variable: stOutputValue
    Rectangle (34,80 42x32), "Min:", text variable: stMin, invisible if: LEN(stMin) = 0
    Rectangle (73,80 157x32), "%s", text variable: stMin, invisible if: LEN(stMin) = 0
    Rectangle (285,80 45x32), "Max:", text variable: stMin, invisible if: LEN(stMax) = 0
    Rectangle (330,80 217x32), "%s", text variable: stMax, invisible if: LEN(stMax) = 0
    Button (20,180 46x54), "´", invisible if: bShift
        OnMouseDown: execute { VisuDlg_CheckedAppend(stOutputValue, stVariableValue, bInit, (flags AND VisuElems.Visu_InputFlags.Password) = 1, '´'); }
    Button (69,180 46x54), "1", invisible if: bShift
        OnMouseDown: execute { VisuDlg_CheckedAppend(stOutputValue, stVariableValue, bInit, (flags AND VisuElems.Visu_InputFlags.Password) = 1, '1'); }
    Button (117,180 46x54), "2", invisible if: bShift
        OnMouseDown: execute { VisuDlg_CheckedAppend(stOutputValue, stVariableValue, bInit, (flags AND VisuElems.Visu_InputFlags.Password) = 1, '2'); }
    Button (166,180 46x54), "3", invisible if: bShift
        OnMouseDown: execute { VisuDlg_CheckedAppend(stOutputValue, stVariableValue, bInit, (flags AND VisuElems.Visu_InputFlags.Password) = 1, '3'); }
    Button (214,180 46x54), "4", invisible if: bShift
        OnMouseDown: execute { VisuDlg_CheckedAppend(stOutputValue, stVariableValue, bInit, (flags AND VisuElems.Visu_InputFlags.Password) = 1, '4'); }
    Button (263,180 46x54), "5", invisible if: bShift
        OnMouseDown: execute { VisuDlg_CheckedAppend(stOutputValue, stVariableValue, bInit, (flags AND VisuElems.Visu_InputFlags.Password) = 1, '5'); }
    Button (311,180 46x54), "6", invisible if: bShift
        OnMouseDown: execute { VisuDlg_CheckedAppend(stOutputValue, stVariableValue, bInit, (flags AND VisuElems.Visu_InputFlags.Password) = 1, '6'); }
    Button (359,180 46x54), "7", invisible if: bShift
        OnMouseDown: execute { VisuDlg_CheckedAppend(stOutputValue, stVariableValue, bInit, (flags AND VisuElems.Visu_InputFlags.Password) = 1, '7'); }
    Button (408,180 46x54), "8", invisible if: bShift
        OnMouseDown: execute { VisuDlg_CheckedAppend(stOutputValue, stVariableValue, bInit, (flags AND VisuElems.Visu_InputFlags.Password) = 1, '8'); }
    Button (456,180 46x54), "9", invisible if: bShift
        OnMouseDown: execute { VisuDlg_CheckedAppend(stOutputValue, stVariableValue, bInit, (flags AND VisuElems.Visu_InputFlags.Password) = 1, '9'); }
    Button (505,180 46x54), "0", invisible if: bShift
        OnMouseDown: execute { VisuDlg_CheckedAppend(stOutputValue, stVariableValue, bInit, (flags AND VisuElems.Visu_InputFlags.Password) = 1, '0'); }
    Button (553,180 46x54), "-", invisible if: bShift
        OnMouseDown: execute { VisuDlg_CheckedAppend(stOutputValue, stVariableValue, bInit, (flags AND VisuElems.Visu_InputFlags.Password) = 1, '-'); }
    Button (601,180 46x54), "=", invisible if: bShift
        OnMouseDown: execute { VisuDlg_CheckedAppend(stOutputValue, stVariableValue, bInit, (flags AND VisuElems.Visu_InputFlags.Password) = 1, '='); }
    Button (570,241 46x54), "{", invisible if: NOT bShift
        OnMouseDown: execute { VisuDlg_CheckedAppend(stOutputValue, stVariableValue, bInit, (flags AND VisuElems.Visu_InputFlags.Password) = 1, '{'); }
    Button (570,241 46x54), "[", invisible if: bShift
        OnMouseDown: execute { VisuDlg_CheckedAppend(stOutputValue, stVariableValue, bInit, (flags AND VisuElems.Visu_InputFlags.Password) = 1, '['); }
    Button (619,241 46x54), "}", invisible if: NOT bShift
        OnMouseDown: execute { VisuDlg_CheckedAppend(stOutputValue, stVariableValue, bInit, (flags AND VisuElems.Visu_InputFlags.Password) = 1, '}'); }
    Button (619,241 46x54), "]", invisible if: bShift
        OnMouseDown: execute { VisuDlg_CheckedAppend(stOutputValue, stVariableValue, bInit, (flags AND VisuElems.Visu_InputFlags.Password) = 1, ']'); }
    Button (667,241 46x54), "\", invisible if: bShift
        OnMouseDown: execute { VisuDlg_CheckedAppend(stOutputValue, stVariableValue, bInit, (flags AND VisuElems.Visu_InputFlags.Password) = 1, '\'); }
    Button (541,303 46x54), ";", invisible if: bShift
        OnMouseDown: execute { VisuDlg_CheckedAppend(stOutputValue, stVariableValue, bInit, (flags AND VisuElems.Visu_InputFlags.Password) = 1, ';'); }
    Button (589,303 46x54), "'", invisible if: bShift
        OnMouseDown: execute { VisuDlg_CheckedAppend(stOutputValue, stVariableValue, bInit, (flags AND VisuElems.Visu_InputFlags.Password) = 1, '$''); }
    Button (474,366 46x54), ",", invisible if: bShift
        OnMouseDown: execute { VisuDlg_CheckedAppend(stOutputValue, stVariableValue, bInit, (flags AND VisuElems.Visu_InputFlags.Password) = 1, ','); }
    Button (522,366 46x54), ".", invisible if: bShift
        OnMouseDown: execute { VisuDlg_CheckedAppend(stOutputValue, stVariableValue, bInit, (flags AND VisuElems.Visu_InputFlags.Password) = 1, '.'); }
    Button (570,366 46x54), "/", invisible if: bShift
        OnMouseDown: execute { VisuDlg_CheckedAppend(stOutputValue, stVariableValue, bInit, (flags AND VisuElems.Visu_InputFlags.Password) = 1, '/'); }
    Button (20,366 112x54), "Shift"
        OnMouseDown: toggle bShift
END_VISUALIZATION

// ---- VISUs/MainFrame.TcVIS
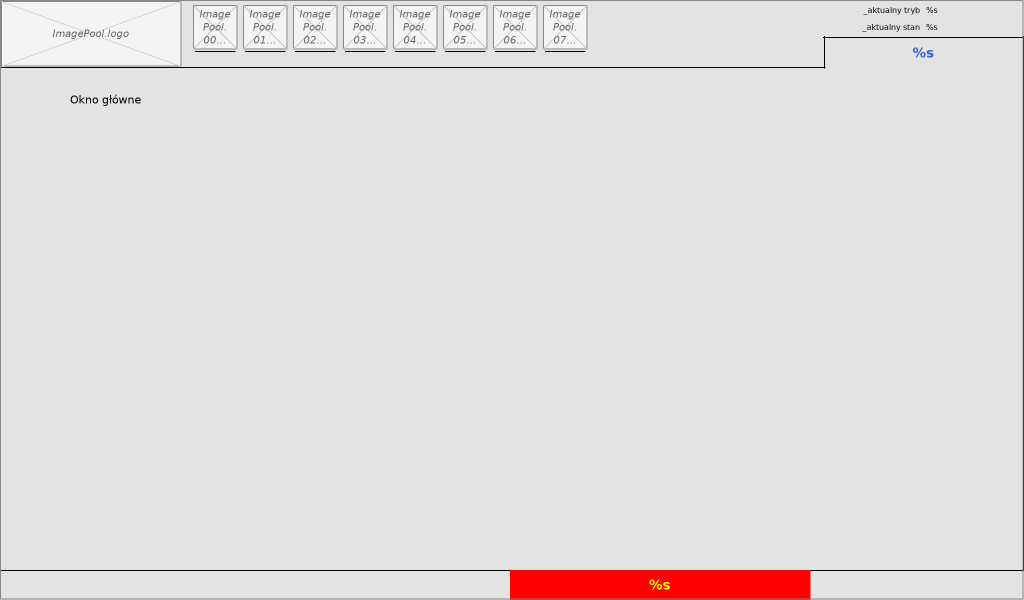
VISUALIZATION MainFrame  // 1024x600
VAR_IN_OUT
	stHMIData		: ST_HMIManager;
END_VAR
    Image (1,1 180x65), image: ImagePool.logo
    Frame (190,5 50x50)
        shows F_MainMenu_00(stMenuButton := stHMIData.stMainMenu.arrButton [0].stButtonHMI)
    Frame (240,5 50x50)
        shows F_MainMenu_01(stMenuButton := stHMIData.stMainMenu.arrButton [1].stButtonHMI)
    Frame (290,5 50x50)
        shows F_MainMenu_02(stMenuButton := stHMIData.stMainMenu.arrButton [2].stButtonHMI)
    Frame (340,5 50x50)
        shows F_MainMenu_03(stMenuButton := stHMIData.stMainMenu.arrButton [3].stButtonHMI)
    Frame (390,5 50x50)
        shows F_MainMenu_04(stMenuButton := stHMIData.stMainMenu.arrButton [4].stButtonHMI)
    Frame (440,5 50x50)
        shows F_MainMenu_05(stMenuButton := stHMIData.stMainMenu.arrButton [5].stButtonHMI)
    Frame (490,5 50x50)
        shows F_MainMenu_06(stMenuButton := stHMIData.stMainMenu.arrButton [6].stButtonHMI)
    Frame (540,5 50x50)
        shows F_MainMenu_07(stMenuButton := stHMIData.stMainMenu.arrButton [7].stButtonHMI)
    Line (0,67) (825,67)
    Line (824,36) (824,68)
    Line (1023,36) (1023,570)
    Line (823,37) (1024,37)
    Line (0,570) (1024,570)
    Line (0,67) (0,570)
    Rectangle (510,570 300x30), "%s", text variable: stHMIData.stMachineControl.stCommonData.stRecipeInformation.wsRecipeInformation, colour variable: stHMIData.stMachineControl.stCommonData.stRecipeInformation.dwBackgroud
        p55702900: stHMIData.stMachineControl.stCommonData.stRecipeInformation.dwText
    Rectangle (827,40 193x26), "%s", text variable: stHMIData.stMainMenu.stMenu.wsTitleActivePage
    Frame (4,71 1015x495), frame switch variable: stHMIData.stMainMenu.stMenu.iNumberOfActivePage
        shows F_00_MainScreen()
        shows F_01_Parameters(stScreenData := stHMIData.stMachineControl.stPrepScr_01_XX)
        shows F_02_Recipe(stScreenData := stHMIData.stMachineControl.stPrepScr_02_XX)
        shows F_03_Events(stScreenData := stHMIData.stMachineControl.stPrepScr_03_XX)
        shows F_04_ChangeMode(stScreenData := stHMIData.stMachineControl.stPrepScr_04_XX)
        shows F_05_Statistics(stScreenData := stHMIData.stMachineControl.stPrepScr_05_XX)
        shows F_06_Diagram(stScreenData := stHMIData.stMachineControl.stPrepScr_06_XX)
        shows F_07_Settings(stScreenData := stHMIData.stMachineControl.stPrepScr_07_XX)
    Rectangle (823,3 100x15), "_aktualny tryb", text list: 'TextListGlobal', text index: 1
    Rectangle (823,20 100x15), "_aktualny stan", text list: 'TextListGlobal', text index: 0
    Rectangle (923,3 100x15), "%s", text variable: stHMIData.stMachineControl.stCommonData.wsActualMode
    Rectangle (923,20 100x15), "%s", text variable: stHMIData.stMachineControl.stCommonData.wsActualState
END_VISUALIZATION

// ---- VISUs/MainMenuFrame/F_00_MainScreen.TcVIS
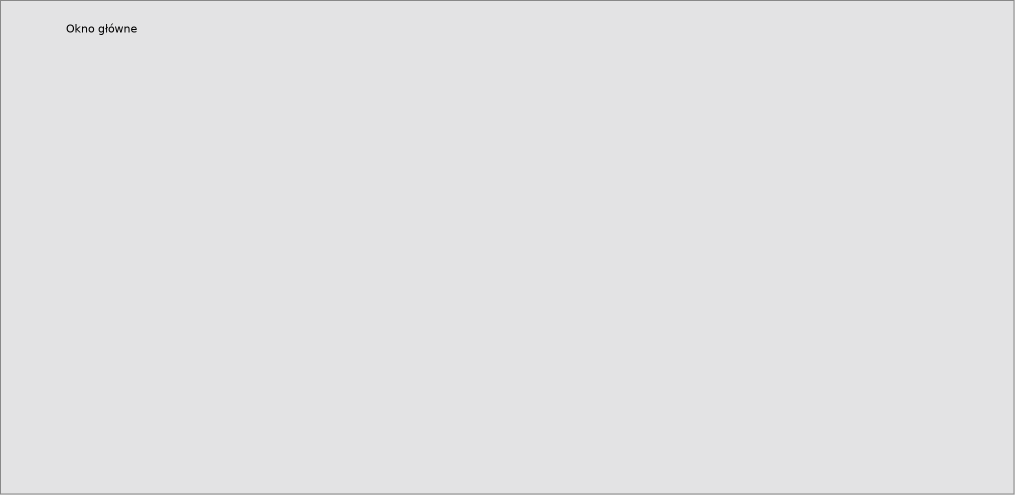
VISUALIZATION F_00_MainScreen  // 1015x495
    Label (27,14 150x30), "Okno główne"
END_VISUALIZATION

// ---- VISUs/MainMenuFrame/F_01_Parameters.TcVIS
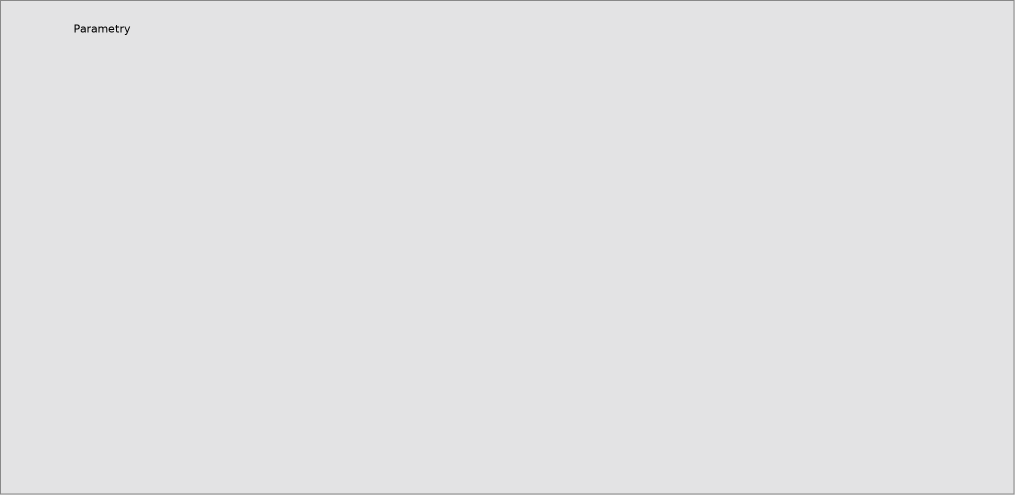
VISUALIZATION F_01_Parameters  // 1015x495
VAR_IN_OUT
	stScreenData	: ST_MCHMIPrepareScreen_01_XX;
	
END_VAR
    Label (27,14 150x30), "Parametry"
END_VISUALIZATION

// ---- VISUs/MainMenuFrame/F_02_Recipe.TcVIS
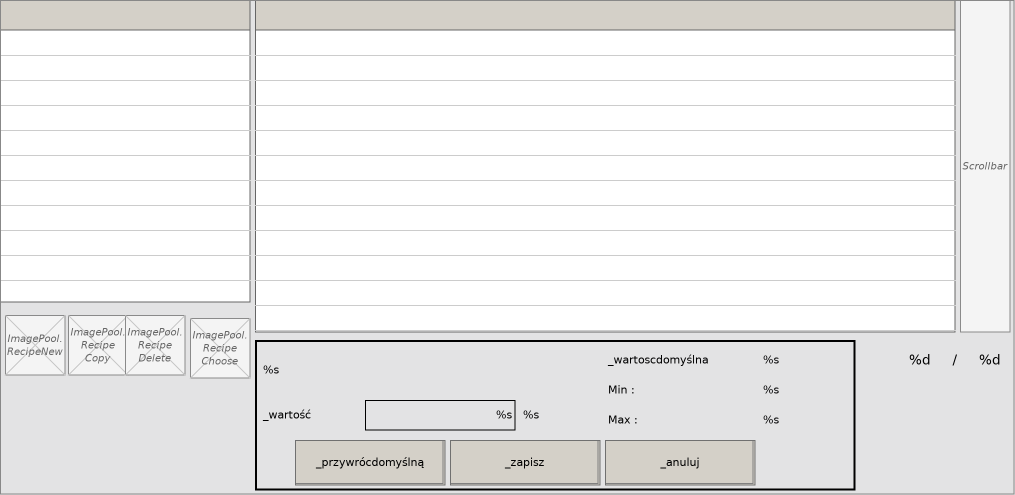
VISUALIZATION F_02_Recipe  // 1015x495
VAR_IN_OUT
	{attribute "VAR_IN_OUT_AS_POINTER}
	stScreenData	: ST_MCHMIPrepareScreen_02_XX;
	
END_VAR
    Table (0,0 250x302), data array: stScreenData.arrNameListRecipe
        p1128707560: stScreenData.iNumberOfRecipe
        p1137915858: stScreenData.iSelectedNameRow
        p1822360349: stScreenData.bSelectedNameRow
        p3854506369: stScreenData.arrNameListRecipe[INDEX]
    Image (5,315 60x60), invisible if: not stScreenData.bVisibleButtonAddFromTemplate, image: ImagePool.RecipeNew
        OnMouseDown: execute { stScreenData.stAddRecipe.bNewRecipeFromTemplate := TRUE; }
        OnMouseUp: OpenDialog Dialog=D_AddRecipe, Parameters={stData: stScreenData.stAddRecipe}, Selected={1: , 2: }, OpenModal=True, OpenCentered=True
    Image (68,315 60x60), invisible if: not stScreenData.bVisibleButtonAddFromRecipe, image: ImagePool.RecipeCopy
        OnMouseDown: execute { stScreenData.stAddRecipe.bNewRecipeFromRecipe := TRUE; }
        OnMouseUp: OpenDialog Dialog=D_AddRecipe, Parameters={stData: stScreenData.stAddRecipe}, Selected={1: , 2: }, OpenModal=True, OpenCentered=True
    Image (125,315 60x60), invisible if: not stScreenData.bVisibleButtonDelete, image: ImagePool.RecipeDelete
        OnMouseDown: execute { stScreenData.stDeleteRecipe.bDeleteRecipe := TRUE; }
        OnMouseUp: OpenDialog Dialog=D_DeleteRecipeCleim, Parameters={stData: stScreenData.stDeleteRecipe}, Selected={1: , 2: }, OpenModal=True, OpenCentered=True
    Image (190,318 60x60), invisible if: not stScreenData.bVisibleButtonChoose, image: ImagePool.RecipeChoose
        OnMouseDown: execute { stScreenData.bSelectRecipe := TRUE; }
    Scrollbar (960,0 50x332), invisible if: not stScreenData.bSelectedNameRow
        p2245068023: stScreenData.stIngredientList.iNumberOfPage
        p1057716461: stScreenData.stIngredientList.iActualPage
    Table (255,0 700x332), invisible if: not stScreenData.bSelectedNameRow, data array: stScreenData.stIngredientList.stList.arrRow
        p3854506369: stScreenData.stIngredientList.stList.arrRow[INDEX].wsText
        p1218418051: stScreenData.stIngredientList.stList.arrRow[INDEX].rDefaultValue
        p2232123230: Opis
        p1128707560: stScreenData.stIngredientList.iNumberRowOnPage
        p4092479075: stScreenData.stIngredientList.stList.arrRow[INDEX].rMin
        p2237128397: stScreenData.stIngredientList.stList.arrRow[INDEX].rMax
        p1137915858: stScreenData.stIngredientList.stList.iSelectedRow
        p1822360349: stScreenData.stIngredientList.stList.bSelectedRow
        p338671338: stScreenData.stIngredientList.stList.arrRow[INDEX].sUnit
        p1755163831: Jednostka
        p1892666644: stScreenData.stIngredientList.stList.arrRow[INDEX].rValue
        p511219082: Wartość
    Group (900,340 110x40), invisible if: not stScreenData.bSelectedNameRow
        Rectangle (0,0 110x40), "/"
        Rectangle (0,0 40x40), "%d", text variable: stScreenData.stIngredientList.iActualPage
        Rectangle (70,0 40x40), "%d", text variable: stScreenData.stIngredientList.iNumberOfPage
    Frame (255,340 600x150), invisible if: not stScreenData.stIngredientList.stList.bSelectedRow
        shows F_Descriptor(stData := stScreenData.stIngredientList.stChossenRow)
END_VISUALIZATION

// ---- VISUs/MainMenuFrame/F_03_Events.TcVIS
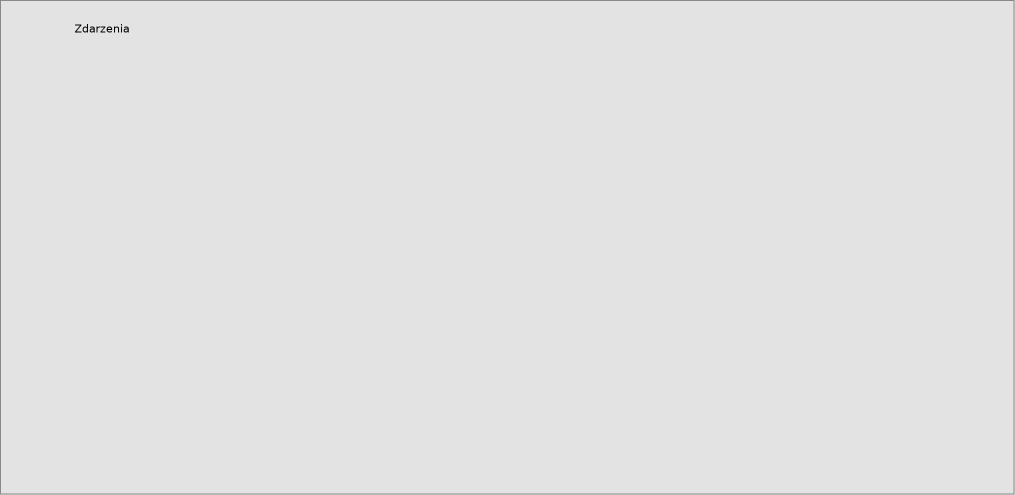
VISUALIZATION F_03_Events  // 1015x495
VAR_IN_OUT
	stScreenData	: ST_MCHMIPrepareScreen_03_XX;
	
END_VAR
    Label (27,14 150x30), "Zdarzenia"
END_VISUALIZATION

// ---- VISUs/MainMenuFrame/F_04_ChangeMode.TcVIS
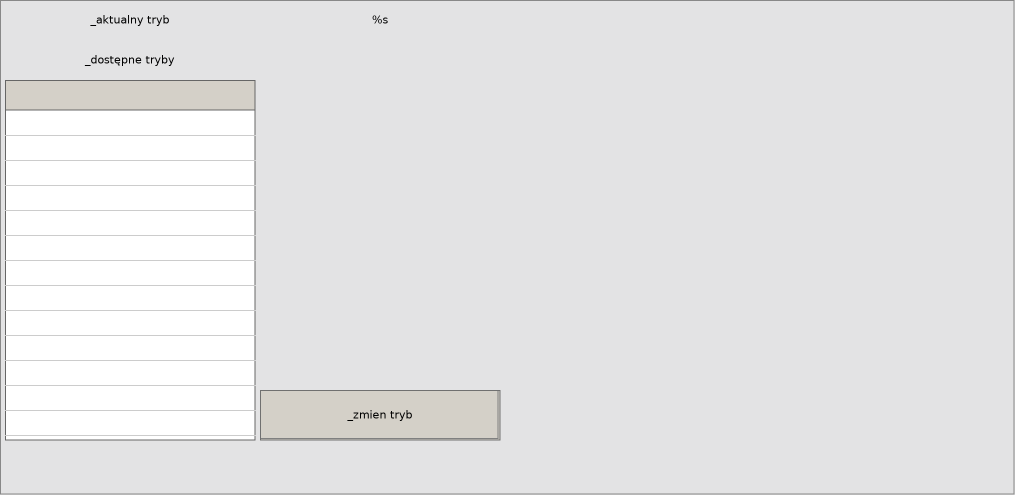
VISUALIZATION F_04_ChangeMode  // 1015x495
VAR_IN_OUT
	stScreenData	: ST_MCHMIPrepareScreen_04_XX;
	
END_VAR
    Rectangle (5,45 250x30), "_dostępne tryby", text list: 'TextList_04', text index: 0
    Table (5,80 250x360), data array: stScreenData.arrNamesOfMode
        p3854506369: stScreenData.arrNamesOfMode[INDEX].wsDescription
        p1892666644: stScreenData.arrNamesOfMode[INDEX].iNumber
        p1128707560: stScreenData.iNumberModeToDisplay-1
        p1137915858: stScreenData.iSelectedMode
        p1822360349: stScreenData.bSelectedRow
    Rectangle (5,5 250x30), "_aktualny tryb", text list: 'TextListGlobal', text index: 1
    Rectangle (255,5 250x30), "%s", text variable: stScreenData.wsActualMode
    Button (260,390 240x50), "_zmien tryb", text list: 'TextList_04', text index: 1
        OnMouseDown: execute { stScreenData.bChangeMode := TRUE; }
END_VISUALIZATION

// ---- VISUs/MainMenuFrame/F_05_Statistics.TcVIS
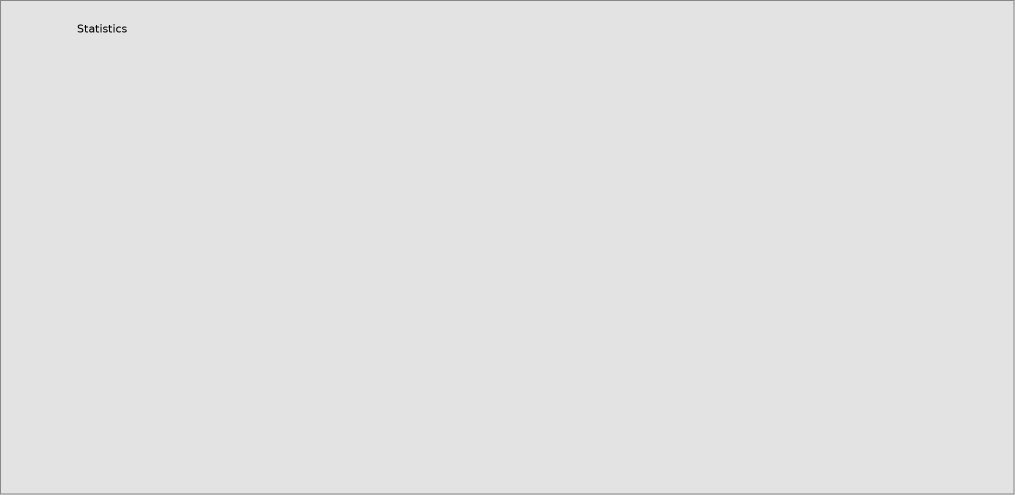
VISUALIZATION F_05_Statistics  // 1015x495
VAR_IN_OUT
	stScreenData	: ST_MCHMIPrepareScreen_05_XX;
	
END_VAR
    Label (27,14 150x30), "Statistics"
END_VISUALIZATION

// ---- VISUs/MainMenuFrame/F_06_Diagram.TcVIS
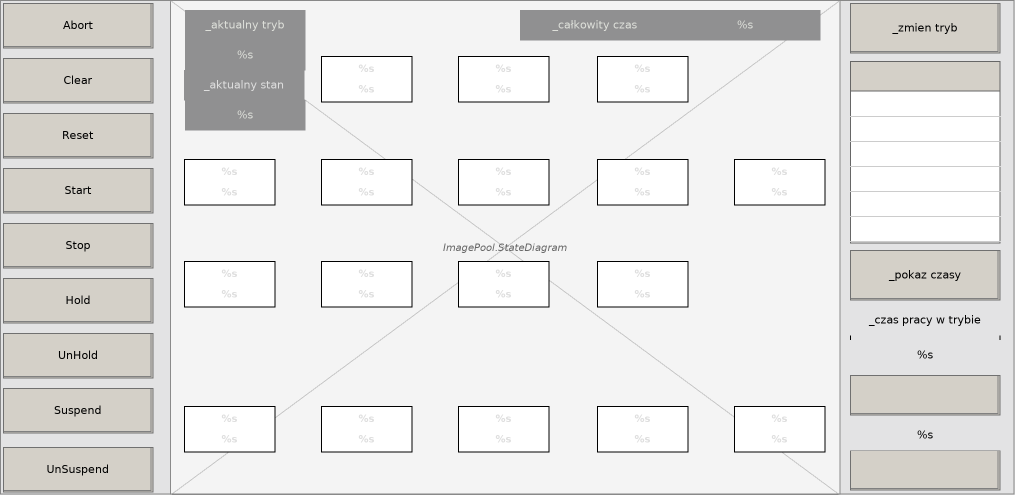
VISUALIZATION F_06_Diagram  // 1015x495
VAR_IN_OUT
	stScreenData	: ST_MCHMIPrepareScreen_06_XX;
	
END_VAR
    Rectangle (540,15 150x65)
    Image (170,0 670x495), image: ImagePool.StateDiagram
    Rectangle (185,10 120x30), "_aktualny tryb", text list: 'TextListGlobal', text index: 1
    Rectangle (185,40 120x30), "%s", text variable: stScreenData.wsActualMode
    Rectangle (184,70 120x30), "_aktualny stan", text list: 'TextListGlobal', text index: 0
    Rectangle (185,100 120x30), "%s", text variable: stScreenData.wsActualState
    Frame (734,406 91x46), invisible if: not stScreenData.arrStateEnabledInMode [1]
        shows F_DiagramState(stStateInfo := stScreenData.arrState [1])
    Frame (597,406 91x46), invisible if: not stScreenData.arrStateEnabledInMode [2]
        shows F_DiagramState(stStateInfo := stScreenData.arrState [2])
    Frame (458,406 91x46), invisible if: not stScreenData.arrStateEnabledInMode [3]
        shows F_DiagramState(stStateInfo := stScreenData.arrState [3])
    Frame (321,406 91x46), invisible if: not stScreenData.arrStateEnabledInMode [4]
        shows F_DiagramState(stStateInfo := stScreenData.arrState [4])
    Frame (184,406 91x46), invisible if: not stScreenData.arrStateEnabledInMode [5]
        shows F_DiagramState(stStateInfo := stScreenData.arrState [5])
    Frame (597,261 91x46), invisible if: not stScreenData.arrStateEnabledInMode [10]
        shows F_DiagramState(stStateInfo := stScreenData.arrState [10])
    Frame (458,261 91x46), invisible if: not stScreenData.arrStateEnabledInMode [11]
        shows F_DiagramState(stStateInfo := stScreenData.arrState [11])
    Frame (321,261 91x46), invisible if: not stScreenData.arrStateEnabledInMode [12]
        shows F_DiagramState(stStateInfo := stScreenData.arrState [12])
    Frame (184,261 91x46), invisible if: not stScreenData.arrStateEnabledInMode [6]
        shows F_DiagramState(stStateInfo := stScreenData.arrState [6])
    Frame (734,159 91x46), invisible if: not stScreenData.arrStateEnabledInMode [17]
        shows F_DiagramState(stStateInfo := stScreenData.arrState [17])
    Frame (597,159 91x46), invisible if: not stScreenData.arrStateEnabledInMode [16]
        shows F_DiagramState(stStateInfo := stScreenData.arrState [16])
    Frame (458,159 91x46), invisible if: not stScreenData.arrStateEnabledInMode [9]
        shows F_DiagramState(stStateInfo := stScreenData.arrState [9])
    Frame (321,159 91x46), invisible if: not stScreenData.arrStateEnabledInMode [8]
        shows F_DiagramState(stStateInfo := stScreenData.arrState [8])
    Frame (184,159 91x46), invisible if: not stScreenData.arrStateEnabledInMode [7]
        shows F_DiagramState(stStateInfo := stScreenData.arrState [7])
    Frame (597,56 91x46), invisible if: not stScreenData.arrStateEnabledInMode [13]
        shows F_DiagramState(stStateInfo := stScreenData.arrState [13])
    Frame (458,56 91x46), invisible if: not stScreenData.arrStateEnabledInMode [14]
        shows F_DiagramState(stStateInfo := stScreenData.arrState [14])
    Frame (321,56 91x46), invisible if: not stScreenData.arrStateEnabledInMode [15]
        shows F_DiagramState(stStateInfo := stScreenData.arrState [15])
    Button (3,58 150x45), "Clear", text list: 'TextList_Opisy'
        OnMouseDown: execute { stScreenData.arrCmdChangeState [E_SaMCommandChangeState.Clear].bPushed := true; }
    Button (3,113 150x45), "Reset", text list: 'TextList_Opisy'
        OnMouseDown: execute { stScreenData.arrCmdChangeState [E_SaMCommandChangeState.Reset].bPushed := true; }
    Button (3,168 150x45), "Start", text list: 'TextList_Opisy'
        OnMouseDown: execute { stScreenData.arrCmdChangeState [E_SaMCommandChangeState.Start].bPushed := true; }
    Button (3,388 150x45), "Suspend", text list: 'TextList_Opisy'
        OnMouseDown: execute { stScreenData.arrCmdChangeState [E_SaMCommandChangeState.Suspend].bPushed := true; }
    Button (3,447 150x45), "UnSuspend", text list: 'TextList_Opisy'
        OnMouseDown: execute { stScreenData.arrCmdChangeState [E_SaMCommandChangeState.Unsuspend].bPushed := true; }
    Button (3,278 150x45), "Hold", text list: 'TextList_Opisy'
        OnMouseDown: execute { stScreenData.arrCmdChangeState [E_SaMCommandChangeState.Hold].bPushed := true; }
    Button (3,333 150x45), "UnHold", text list: 'TextList_Opisy'
        OnMouseDown: execute { stScreenData.arrCmdChangeState [E_SaMCommandChangeState.Unhold].bPushed := true; }
    Button (3,3 150x45), "Abort"
        OnMouseDown: execute { stScreenData.arrCmdChangeState [E_SaMCommandChangeState.Abort ].bPushed := true; }
    Button (3,223 150x45), "Stop", text list: 'TextList_Opisy'
        OnMouseDown: execute { stScreenData.arrCmdChangeState [E_SaMCommandChangeState.Stop].bPushed := true; }
    Rectangle (520,10 150x30), "_całkowity czas", text list: 'TextList_06', text index: 0
    Rectangle (670,10 150x30), "%s", text variable: stScreenData.sTotalWorkTime
    Button (850,3 150x50), "_zmien tryb", text list: 'TextList_06', text index: 1
        OnMouseDown: execute { stScreenData.bChangeMode := TRUE; }
    Button (850,250 150x50), "_pokaz czasy", text list: 'TextList_06', text index: 2
        toggle stScreenData.bShowTime
    Rectangle (850,305 150x65), invisible if: not stScreenData.bShowTime
    Rectangle (850,305 150x30), "_czas pracy w trybie", invisible if: not stScreenData.bShowTime, text list: 'TextList_06', text index: 3
    Rectangle (850,340 150x30), "%s", text variable: stScreenData.sWorkingTimeInMode, invisible if: not stScreenData.bShowTime
    Button (850,375 150x40), invisible if: not stScreenData.bShowTime, text list: 'TextList_06', text index: 4
        OnMouseDown: execute { stScreenData.bNextModeToDisplayTime := TRUE; }
    Button (850,450 150x40), invisible if: not stScreenData.bShowTime, text list: 'TextList_06', text index: 5
        OnMouseDown: execute { stScreenData.bPrevModeToDisplayTime := TRUE; }
    Rectangle (850,420 150x30), "%s", text variable: stScreenData.wsNameModeOfTimeDisplay, invisible if: not stScreenData.bShowTime
    Table (850,61 150x182), data array: stScreenData.arrNamesOfMode
        p3854506369: stScreenData.arrNamesOfMode[INDEX].wsDescription
        p1892666644: stScreenData.arrNamesOfMode[INDEX].iNumber
        p1128707560: stScreenData.iNumberModeToDisplay-1
        p1137915858: stScreenData.iSelectedMode
        p1822360349: stScreenData.bSelectedRow
END_VISUALIZATION

// ---- VISUs/MainMenuFrame/F_07_Settings.TcVIS
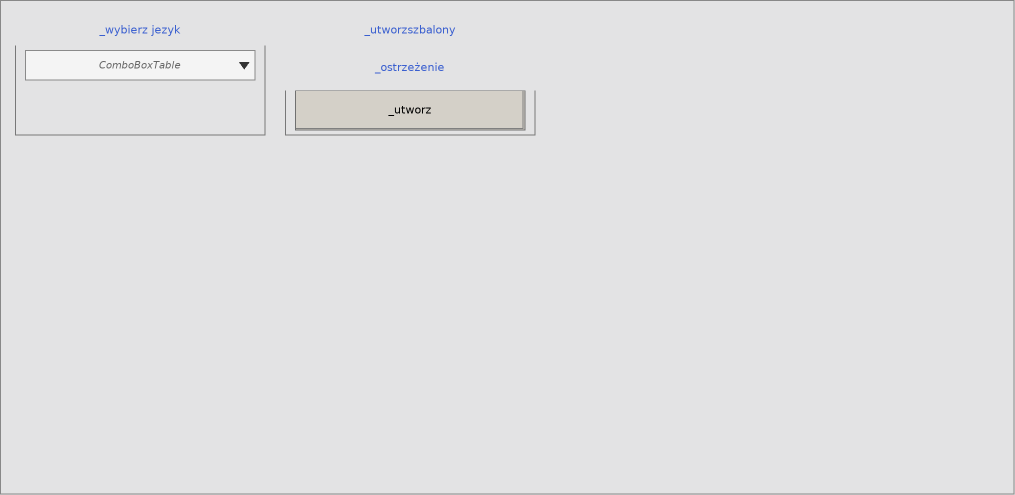
VISUALIZATION F_07_Settings  // 1015x495
VAR_IN_OUT
	stScreenData	: ST_MCHMIPrepareScreen_07_XX;

END_VAR
    Rectangle (15,15 250x120)
    Rectangle (15,15 250x30), "_wybierz jezyk", text list: 'TextList_07', text index: 0
    ComboBoxTable (25,50 230x30), variable: stScreenData.iChoosoLocation, data array: stScreenData.arrLocationDescription
        p3854506369: stScreenData.arrLocationDescription[INDEX]
        p1128707560: GVL_BaseConstans.NUMBER_OF_LOCATIONS -1
    Rectangle (285,15 250x120)
    Rectangle (285,15 250x30), "_utworzszbalony", text list: 'TextList_07', text index: 1
    Button (295,90 230x40), "_utworz", text list: 'TextList_07', text index: 3
        OnMouseDown: execute { stScreenData.bCreateRecipeTemplate := TRUE; }
    Rectangle (285,45 250x45), "_ostrzeżenie", text list: 'TextList_07', text index: 2
END_VISUALIZATION

// ---- VISUs/MainMenu/F_MainMenu_00.TcVIS
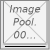
VISUALIZATION F_MainMenu_00  // 50x50
VAR_IN_OUT
	stMenuButton	: ST_HMIEButton_HMI;
END_VAR
    Image (3,0 44x44), invisible if: not stMenuButton.bVisible, image: ImagePool.00_MainScreen
        OnMouseDown: execute { stMenuButton.bPushed := TRUE; }
    Line (5,46) (45,46), invisible if: not stMenuButton.bVisible or not stMenuButton.bActive, input disabled if: not stMenuButton.bEnable
END_VISUALIZATION

// ---- VISUs/MainMenu/F_MainMenu_01.TcVIS
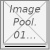
VISUALIZATION F_MainMenu_01  // 50x50
VAR_IN_OUT
	stMenuButton	: ST_HMIEButton_HMI;
END_VAR
    Image (3,0 44x44), invisible if: not stMenuButton.bVisible, image: ImagePool.01_Parameters
        OnMouseDown: execute { stMenuButton.bPushed := TRUE; }
    Line (5,46) (45,46), invisible if: not stMenuButton.bVisible or not stMenuButton.bActive, input disabled if: not stMenuButton.bEnable
END_VISUALIZATION

// ---- VISUs/MainMenu/F_MainMenu_02.TcVIS
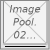
VISUALIZATION F_MainMenu_02  // 50x50
VAR_IN_OUT
	stMenuButton	: ST_HMIEButton_HMI;
END_VAR
    Image (3,0 44x44), invisible if: not stMenuButton.bVisible, image: ImagePool.02_Recipe
        OnMouseDown: execute { stMenuButton.bPushed := TRUE; }
    Line (5,46) (45,46), invisible if: not stMenuButton.bVisible or not stMenuButton.bActive, input disabled if: not stMenuButton.bEnable
END_VISUALIZATION

// ---- VISUs/MainMenu/F_MainMenu_03.TcVIS
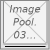
VISUALIZATION F_MainMenu_03  // 50x50
VAR_IN_OUT
	stMenuButton	: ST_HMIEButton_HMI;
END_VAR
    Image (3,0 44x44), invisible if: not stMenuButton.bVisible, image: ImagePool.03_Events
        OnMouseDown: execute { stMenuButton.bPushed := TRUE; }
    Line (5,46) (45,46), invisible if: not stMenuButton.bVisible or not stMenuButton.bActive, input disabled if: not stMenuButton.bEnable
END_VISUALIZATION

// ---- VISUs/MainMenu/F_MainMenu_04.TcVIS
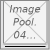
VISUALIZATION F_MainMenu_04  // 50x50
VAR_IN_OUT
	stMenuButton	: ST_HMIEButton_HMI;
END_VAR
    Image (3,0 44x44), invisible if: not stMenuButton.bVisible, image: ImagePool.04_ChangeMode
        OnMouseDown: execute { stMenuButton.bPushed := TRUE; }
    Line (5,46) (45,46), invisible if: not stMenuButton.bVisible or not stMenuButton.bActive, input disabled if: not stMenuButton.bEnable
END_VISUALIZATION

// ---- VISUs/MainMenu/F_MainMenu_05.TcVIS
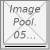
VISUALIZATION F_MainMenu_05  // 50x50
VAR_IN_OUT
	stMenuButton	: ST_HMIEButton_HMI;
END_VAR
    Image (3,0 44x44), invisible if: not stMenuButton.bVisible, image: ImagePool.05_Statistics
        OnMouseDown: execute { stMenuButton.bPushed := TRUE; }
    Line (5,46) (45,46), invisible if: not stMenuButton.bVisible or not stMenuButton.bActive, input disabled if: not stMenuButton.bEnable
END_VISUALIZATION

// ---- VISUs/MainMenu/F_MainMenu_06.TcVIS
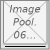
VISUALIZATION F_MainMenu_06  // 50x50
VAR_IN_OUT
	stMenuButton	: ST_HMIEButton_HMI;
END_VAR
    Image (3,0 44x44), invisible if: not stMenuButton.bVisible, image: ImagePool.06_Diagram
        OnMouseDown: execute { stMenuButton.bPushed := TRUE; }
    Line (5,46) (45,46), invisible if: not stMenuButton.bVisible or not stMenuButton.bActive, input disabled if: not stMenuButton.bEnable
END_VISUALIZATION

// ---- VISUs/MainMenu/F_MainMenu_07.TcVIS
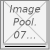
VISUALIZATION F_MainMenu_07  // 50x50
VAR_IN_OUT
	stMenuButton	: ST_HMIEButton_HMI;
END_VAR
    Image (3,0 44x44), invisible if: not stMenuButton.bVisible, image: ImagePool.07_Setings
        OnMouseDown: execute { stMenuButton.bPushed := TRUE; }
    Line (5,46) (45,46), invisible if: not stMenuButton.bVisible or not stMenuButton.bActive, input disabled if: not stMenuButton.bEnable
END_VISUALIZATION

// ---- VISUs/TextListFrame/TextList_00.TcTLO
TEXTLIST TextList_00
   = ''
END_TEXTLIST

// ---- VISUs/TextListFrame/TextList_01.TcTLO
TEXTLIST TextList_01
   = ''
END_TEXTLIST

// ---- VISUs/TextListFrame/TextList_02.TcTLO
TEXTLIST TextList_02
  0 = 'Czy napewno usunąć recepturę ?' | pl: 'Czy napewno usunąć recepturę ?' | en: 'Are you sure you want to delete the recipe?' | de: 'Möchten Sie das Rezept wirklich löschen?'
   = ''
END_TEXTLIST

// ---- VISUs/TextListFrame/TextList_03.TcTLO
TEXTLIST TextList_03
   = ''
END_TEXTLIST

// ---- VISUs/TextListFrame/TextList_04.TcTLO
TEXTLIST TextList_04
  0 = 'Dostępne tryby pracy' | pl: 'Dostępne tryby pracy' | en: 'Available operating modes' | de: 'Verfügbare Betriebsmodi'
  1 = 'Zmień tryb' | pl: 'Zmień tryb' | en: 'Change mode' | de: 'Modus ändern'
   = ''
END_TEXTLIST

// ---- VISUs/TextListFrame/TextList_05.TcTLO
TEXTLIST TextList_05
   = ''
END_TEXTLIST

// ---- VISUs/TextListFrame/TextList_06.TcTLO
TEXTLIST TextList_06
  0 = 'Całkowity czas' | pl: 'Całkowity czas' | en: 'Total time' | de: 'Gesamtzeit'
  1 = 'Zmień tryb' | pl: 'Zmień tryb' | en: 'Change mode' | de: 'Modus ändern'
  2 = 'Pokaż czasy' | pl: 'Pokaż czasy' | en: 'Show times' | de: 'Zeiten anzeigen'
  3 = 'Czas pracy w trybie' | pl: 'Czas pracy w trybie' | en: 'Working time in mode' | de: 'Arbeitszeit im Modus'
  4 = 'Zmień tryb\nw górę' | pl: 'Zmień tryb\nw górę' | en: 'Change mode\nup' | de: 'Change mode\nup'
  5 = 'Zmień tryb\nw dół' | pl: 'Zmień tryb\nw dół' | en: 'Change mode\ndown' | de: 'Modus ändern\nunten'
   = ''
END_TEXTLIST

// ---- VISUs/TextListFrame/TextList_07.TcTLO
TEXTLIST TextList_07
  0 = 'Wybierz język' | pl: 'Wybierz język' | en: 'Select language' | de: 'Sprache auswählen'
  1 = 'Utwórz szablon receptur' | pl: 'Utwórz szablon receptur' | en: 'Create a recipe template' | de: 'Erstellen Sie eine Rezeptvorlage'
  2 = 'Utworzenie szablonów spowoduje usunięcie istniejących receptur' | pl: 'Utworzenie szablonów spowoduje usunięcie istniejących receptur' | en: 'Creating templates will delete existing recipes' | de: 'Beim Erstellen von Vorlagen werden bestehende Rezepte gelöscht.'
  3 = 'Utwórz' | pl: 'Utwórz' | en: 'Create' | de: 'Erstellen'
   = ''
END_TEXTLIST

// ---- VISUs/TextListGlobal.TcTLO
TEXTLIST TextListGlobal
  0 = 'Aktualny stan : ' | pl: 'Aktualny stan : ' | en: 'Current state : ' | de: 'Aktueller Zustand : '
  1 = 'Aktualny tryb : ' | pl: 'Aktualny tryb : ' | en: 'Current mode : ' | de: 'Aktueller Modus : '
  2 = 'Anuluj' | pl: 'Anuluj' | en: 'Cancel' | de: 'Stornieren'
  3 = 'Przywróc domyślną wartość' | pl: 'Przywróc domyślną wartość' | en: 'Restore default value' | de: 'Standardwert wiederherstellen'
  4 = 'Zapisz' | pl: 'Zapisz' | en: 'Save' | de: 'Speichern'
  5 = 'Wartość domyślna' | pl: 'Wartość domyślna' | en: 'Default value' | de: 'Standardwert'
  6 = 'Wartość' | pl: 'Wartość' | en: 'Value' | de: 'Wert'
  7 = 'Brak wybranej receptury' | pl: 'Brak wybranej receptury' | en: 'No recipe selected' | de: 'Kein Rezept ausgewählt'
   = ''
END_TEXTLIST

// ---- VISUs/Visualization.TcVIS
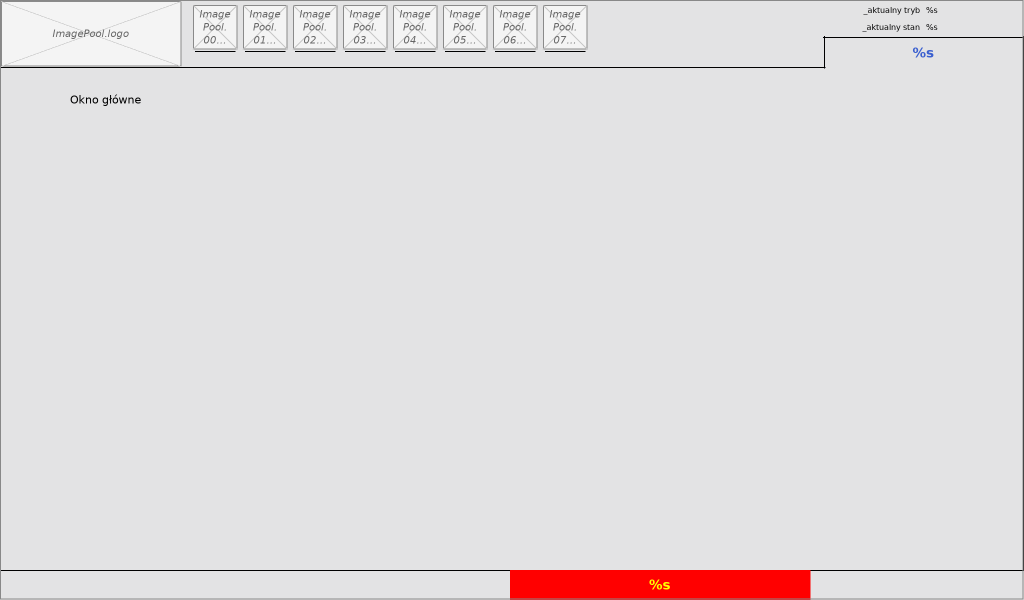
VISUALIZATION Visualization  // 1024x600
    Frame (0,0 1024x600)
        shows MainFrame(stHMIData := MAIN.stDataHMI)
END_VISUALIZATION
